(* CODESYS project CODESYS_BLOG_OPCUA_Part1.project

Project tree, tasks and I/O mapping:
  Device : CODESYS Control Win V3 x64, 3S - Smart Software Solutions GmbH, version 3.5.12.0
    application Application
      task MainTask (cyclic, interval t#20ms, priority 1) calls PLC_PRG
      program PLC_PRG [ST]
      global variables GVL
      Symbols
*)

// Device/Application/GVL
{attribute 'qualified_only'}
VAR_GLOBAL
	uiCycleCounter:INT:=1;
	sInfoMsg:STRING:='INFO: Running';
END_VAR

// Device/Application/PLC_PRG
PROGRAM PLC_PRG
VAR
END_VAR

GVL.uiCycleCounter;
GVL.sInfoMsg;

END_PROGRAM
